(* IEC 61131-3 sources: ecmc_plugin_strucpp/examples/psi_ioc_examples/ioc_project_example/src, 2 files *)

(* ---- main_counter_fb.st ---- *)
FUNCTION_BLOCK COUNTER_FB
VAR_INPUT
  Enable : BOOL;
END_VAR
VAR_OUTPUT
  Value : INT;
END_VAR

IF Enable THEN
  Value := Value + 1;
ELSE
  Value := 0;
END_IF;
END_FUNCTION_BLOCK

(* ---- main.st ---- *)
PROGRAM MAIN
VAR
  actual_position    AT %IW0 : INT;   // @ecmc ec.s14.positionActual01
  drive_control      AT %QW0 : WORD;  // @ecmc ec.s14.driveControl01
  velocity_setpoint  AT %QW2 : INT;   // @ecmc ec.s14.velocitySetpoint01
  cycle_counter      AT %MW0 : INT;   // @epics rec=Main-CycleCounterAct
  manual_velocity             : INT;   // @epics rw rec=Main-ManualVelocity-RB
  actual_pos_export           : INT;   // @epics prefix=$(IOC): rec=Main-PosActCustom
  counter_fb                  : COUNTER_FB;
END_VAR

actual_pos_export := actual_position;
drive_control := 16#0001;
counter_fb(Enable := TRUE);
cycle_counter := counter_fb.Value;

IF manual_velocity <> 0 THEN
  velocity_setpoint := manual_velocity;
ELSIF actual_position < 1000 THEN
  velocity_setpoint := 1000;
ELSE
  velocity_setpoint := -1000;
END_IF;
END_PROGRAM
